TYPE ST_FeedbackQualisys :
STRUCT
	status : DINT := -1;
	d : REAL;
	x : REAL;
	y : REAL;
	z : REAL;
END_STRUCT
END_TYPE

(* stored: Version 1.1.0.1, ProductVersion 3.1.4022.7
   DUT ST_FeedbackQualisys: Id {756fa40c-3d23-4fbc-adc0-4f5d1d624e97} *)
